// TIA Portal V18 export
DATA_BLOCK "L1_tracking"   // DB30
{ S7_Optimized_Access := 'TRUE' }
VERSION : 0.1
// stored: AutoNumber false, DBAccessibleFromOPCUA true, DBAccessibleFromWebserver true, IsOnlyStoredInLoadMemory false, IsRetainMemResEnabled false, IsWriteProtectedInAS false, MemoryReserve 100
   VAR RETAIN
      tracking : Array[1.."N_STAZIONI"] of "LGasp_typeTracking";
   END_VAR
   VAR
      tracking_null : "LGasp_typeTracking";
      reset : Int;   // Indica l'indice della stazione da resettare
   END_VAR
BEGIN
   // tracking[1].info.num_pezzo : Numero pezzo: Ex "tracking_id"
   // tracking[1].info.tipologia : Tipo di profilo: Ex "profile_id"
   // tracking[1].info.nome_articolo : nome articolo: Ex "article"
   // tracking[1].info.lotto : nome lotto: rimasto invariato
   // tracking[1].info.ID_riga : ID riga: Ex "lotto_id"
   // tracking[1].info.lunghezza : lunghezza [mm]: Ex "lenght"
   // tracking[1].info.larghezza : larghezza [mm]: Ex "width"
   // tracking[1].info.altezza : altezza [mm]: Ex "height"
   // tracking[1].info.spessore : spessore [mm]: Ex "thickness"
   // tracking[1].info.testo_stampa : testo da stampare: rimasto invariato
   // tracking[1].info.layout_stampa : layout da impostare: rimasto invariato
   // tracking[1].info.qualita_pezzo : qualità del pezzo (buono, seconda scelta, scarto): Ex "Wastepiece"
END_DATA_BLOCK
